FUNCTION CheckDivWord : WORD
VAR_INPUT
    divisor : WORD;
END_VAR
VAR
END_VAR

IF divisor = 0 THEN
    CheckDivWord := 1;
ELSE
    CheckDivWord := divisor;
END_IF

END_FUNCTION

(* stored: Version 1.1.0.1, ProductVersion 3.1.4024.12
   POU CheckDivWord: Id {a45df642-5814-40a6-801b-e0a8b9fb4517}, SpecialFunc None *)
